FUNCTION_BLOCK NumericValue_PHYS (* Input service interface function block — outputs physical REAL value via NumericObjectPool_S (scale/offset applied in software) *)
  (* Standard: ISO 11783-6; Description: Copyright (c) 2026 Meisterschulen am Ostbahnhof This program and the accompanying materials are made available under the terms of the Eclipse Public License 2.0 which is available at https://www.eclipse.org/legal/epl-2.0/ SPDX-License-Identifier: EPL-2.0 *)
  (* Version 1.0, 2026-04-14, Franz Höpfinger, Meisterschulen am Ostbahnhof, initial API and implementation and/or initial documentation *)
  PACKAGE isobus::UT::io::NumericValue;
  IMPORT logiBUS::utils::conversion::phys::NumericObjectPool_S;
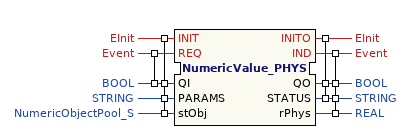
  EVENT_INPUT
    INIT : EInit WITH QI, PARAMS, stObj; (* Service Initialization *)
    REQ WITH QI; (* Service Request *)
  END_EVENT
  EVENT_OUTPUT
    INITO : EInit WITH QO, STATUS; (* Initialization Confirm *)
    IND WITH QO, STATUS, rPhys; (* Indication from Resource *)
  END_EVENT
  VAR_INPUT
    QI : BOOL; (* Event Input Qualifier *)
    PARAMS : STRING; (* Service Parameters *)
    stObj : logiBUS::utils::conversion::phys::NumericObjectPool_S; (* Object pool properties (u16ObjId, scale, offset, decimals) *)
  END_VAR
  VAR_OUTPUT
    QO : BOOL; (* Event Output Qualifier *)
    STATUS : STRING; (* Service Status *)
    rPhys : REAL; (* Physical value (scale/offset applied via stObj) *)
  END_VAR
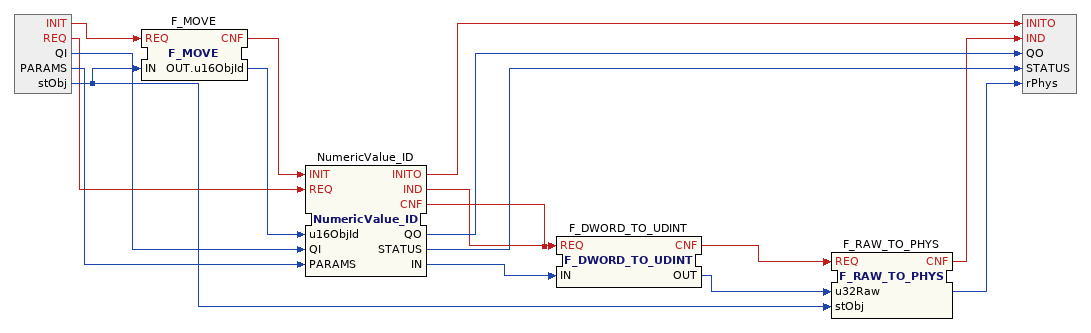
  FBS
    NumericValue_ID : isobus::UT::io::NumericValue::NumericValue_ID;
    F_DWORD_TO_UDINT : iec61131::conversion::F_DWORD_TO_UDINT;
    F_RAW_TO_PHYS : logiBUS::utils::conversion::phys::F_RAW_TO_PHYS;
    F_MOVE : iec61131::selection::F_MOVE; {SET_ATTRIBUTE(DataType, logiBUS::utils::conversion::phys::NumericObjectPool_S)}
  END_FBS
  EVENT_CONNECTIONS
    INIT TO F_MOVE.REQ;
    F_MOVE.CNF TO NumericValue_ID.INIT;
    REQ TO NumericValue_ID.REQ;
    NumericValue_ID.INITO TO INITO;
    NumericValue_ID.IND TO F_DWORD_TO_UDINT.REQ;
    NumericValue_ID.CNF TO F_DWORD_TO_UDINT.REQ;
    F_DWORD_TO_UDINT.CNF TO F_RAW_TO_PHYS.REQ;
    F_RAW_TO_PHYS.CNF TO IND;
  END_CONNECTIONS
  DATA_CONNECTIONS
    stObj TO F_MOVE.IN;
    F_MOVE.OUT.u16ObjId TO NumericValue_ID.u16ObjId;
    QI TO NumericValue_ID.QI;
    PARAMS TO NumericValue_ID.PARAMS;
    NumericValue_ID.QO TO QO;
    NumericValue_ID.STATUS TO STATUS;
    NumericValue_ID.IN TO F_DWORD_TO_UDINT.IN;
    F_DWORD_TO_UDINT.OUT TO F_RAW_TO_PHYS.u32Raw;
    stObj TO F_RAW_TO_PHYS.stObj;
    F_RAW_TO_PHYS. TO rPhys;
  END_CONNECTIONS
END_FUNCTION_BLOCK
